{attribute 'to_string'}
TYPE E_Axis : (
		Master := 0,
		Slave
	);
END_TYPE

(* stored: Version 1.1.0.1
   DUT E_Axis: Id {1c7e21b2-ac77-4006-ae61-8f7091cd5b07} *)
